PROGRAM P_Test
VAR
	
nAngle : LREAL;
nAngle_decimal : int;
nAngle_Final : LREAL;
sWriteFromHMI : STRING;
sWriteToHMI : STRING:='This Is From PLC';
b_HMI_StartLine : BOOL;
b_HMI_StopLine : BOOL;
bStartTrig: R_TRIG;
bStopTrig: R_TRIG;

bSpeedInc		:BOOL;
bSpeedDecrease  :BOOL;
stStatus		:STRING;
// State
n : INT;
END_VAR


bStartTrig(CLK:=b_HMI_StartLine , Q=> );
bStopTrig(CLK:=b_HMI_StopLine , Q=> );

IF ( stStatus='' OR stStatus='Stopped') 
	AND bStartTrig.Q THEN
	stStatus:='Started';

END_IF

IF stStatus='Started' AND bStopTrig.Q THEN
	stStatus:='Stopped';
	nAngle :=0;
END_IF

IF  stStatus='Started' THEN
	
	IF nAngle<180 THEN
		nAngle :=nAngle+0.01;
	END_IF
	//nAngle_decimal:=find((LREAL_TO_STRING(nAngle)),'.');
		
	IF nAngle>=180 THEN
		nAngle :=0;
	END_IF
END_IF
nAngle_Final :=LREAL_TO_UINT(STRING_TO_LREAL(left((LREAL_TO_STRING(nAngle)),((find((LREAL_TO_STRING(nAngle)),'.'))+2))));

END_PROGRAM

(* stored: Version 1.1.0.1, ProductVersion 3.1.4024.12
   POU P_Test: Id {cb104a88-10ac-412f-bdbc-3e45b7e608e4}, SpecialFunc None *)
